// TIA Portal V15.1 export
// export: Created 2020-06-12T07:35:44.7412109Z, ExportSetting None, DisplayName Totally Integrated Automation Portal, DisplayVersion V15.1, DisplayName TIA Portal Openness, DisplayVersion V15.1, DisplayName STEP 7 Professional, DisplayVersion V15.1, DisplayName STEP 7 Safety, DisplayVersion V15.1, DisplayName WinCC Advanced, DisplayVersion V15.1
DATA_BLOCK "VIS_MSG_DB"   // DB812
{ S7_Optimized_Access := 'TRUE' }
// stored: MemoryReserve 100
   VAR RETAIN
      emer : "VISU_MSG";   // Emergency line is not ok
      volt : "VISU_MSG";   // Control voltage trip
      lev_tnk : "VISU_MSG";   // CW Tank level is low
      prs_mod : "VISU_MSG";   // CW module pressure is low
      epump : "VISU_MSG";   // CW emergency pump is ON
      pump_stop : "VISU_MSG";   // CW Pumps problem
      tnk_leak : "VISU_MSG";   // CW Tank leakage
      cw_emer : "VISU_MSG";   // CW Emergency water is open
      cw_filter : "VISU_MSG";   // CW filter is clogged
      acool1 : "VISU_MSG";   // Aftercooling time MS1 is over
      acool2 : "VISU_MSG";   // Aftercooling time MS2 is over
      ecar_near : "VISU_MSG";   // Electrode carriage near bottom position
      ecar_bot : "VISU_MSG";   // Electrode carriage in bottom position
      ht_near : "VISU_MSG";   // Hottopping starts in 1 minute
      alloy1 : "VISU_MSG";   // Alloy bin 1 is empty
      alloy2 : "VISU_MSG";   // Alloy bin 2 is empty
      alloy3 : "VISU_MSG";   // Alloy bin 3 is empty
      lime_empty : "VISU_MSG";
   END_VAR
BEGIN
   emer.in := FALSE;
   emer.ack := FALSE;
   emer.out := TRUE;
   emer.fl := FALSE;
   volt.in := FALSE;
   volt.ack := FALSE;
   volt.out := FALSE;
   volt.fl := FALSE;
   lev_tnk.in := FALSE;
   lev_tnk.ack := FALSE;
   lev_tnk.out := TRUE;
   lev_tnk.fl := FALSE;
   prs_mod.in := FALSE;
   prs_mod.ack := FALSE;
   prs_mod.out := TRUE;
   prs_mod.fl := FALSE;
   epump.in := FALSE;
   epump.ack := FALSE;
   epump.out := FALSE;
   epump.fl := FALSE;
   pump_stop.in := FALSE;
   pump_stop.ack := FALSE;
   pump_stop.out := TRUE;
   pump_stop.fl := FALSE;
   tnk_leak.in := FALSE;
   tnk_leak.ack := FALSE;
   tnk_leak.out := TRUE;
   tnk_leak.fl := FALSE;
   cw_emer.in := FALSE;
   cw_emer.ack := FALSE;
   cw_emer.out := TRUE;
   cw_emer.fl := FALSE;
   cw_filter.in := FALSE;
   cw_filter.ack := FALSE;
   cw_filter.out := FALSE;
   cw_filter.fl := FALSE;
   acool1.in := TRUE;
   acool1.ack := FALSE;
   acool1.out := TRUE;
   acool1.fl := TRUE;
   acool2.in := FALSE;
   acool2.ack := FALSE;
   acool2.out := TRUE;
   acool2.fl := FALSE;
   ecar_near.in := FALSE;
   ecar_near.ack := FALSE;
   ecar_near.out := FALSE;
   ecar_near.fl := FALSE;
   ecar_bot.in := FALSE;
   ecar_bot.ack := FALSE;
   ecar_bot.out := FALSE;
   ecar_bot.fl := FALSE;
   ht_near.in := FALSE;
   ht_near.ack := FALSE;
   ht_near.out := TRUE;
   ht_near.fl := FALSE;
   alloy1.in := FALSE;
   alloy1.ack := FALSE;
   alloy1.out := FALSE;
   alloy1.fl := FALSE;
   alloy2.in := FALSE;
   alloy2.ack := FALSE;
   alloy2.out := FALSE;
   alloy2.fl := FALSE;
   alloy3.in := FALSE;
   alloy3.ack := FALSE;
   alloy3.out := FALSE;
   alloy3.fl := FALSE;
   lime_empty.in := FALSE;
   lime_empty.ack := FALSE;
   lime_empty.out := FALSE;
   lime_empty.fl := FALSE;
END_DATA_BLOCK
